INTERFACE IGenerator

METHOD Flash : BOOL
VAR_INPUT
END_VAR
END_METHOD

PROPERTY P_tCycleTime : Time
GET
END_GET
SET
END_SET
END_PROPERTY

PROPERTY P_Vendor : string
GET
END_GET
END_PROPERTY

END_INTERFACE

(* stored: Version 1.1.0.1, ProductVersion 3.1.4022.16
   Itf IGenerator: Id {2fbe3278-bc5d-4122-9eef-eb57cf51c55d}
   Method Flash: Id {c7ebeb46-d650-40d0-b3ee-dc611a747ad4}
   Property P_tCycleTime: Id {8be20884-2d84-4af2-99c4-ec9fd4841885}
   Get Get: Id {180e54dd-a544-4a11-bf37-7e054aa0bbee}
   Set Set: Id {914010a1-c540-46a0-9f61-2e1a846e3d6d}
   Property P_Vendor: Id {2ff79cf1-4fe2-47c0-a9db-bf46f5ba5790}
   Get Get: Id {c72fe078-5b97-4e6e-a8a5-03cef3c34f72} *)
